FUNCTION_BLOCK RobotA26 EXTENDS KukaRobot
VAR_INPUT
	conveyorSafety : BOOL;
END_VAR
VAR_OUTPUT //from outputs array
	{warning disable C0195}
	taskID : TaskA26;
	param1 : INT; //position number (1..6)
	param2 : INT;
	
	strapSafetyOut : BOOL;
END_VAR
VAR_OUTPUT //from inputs array
	tool : SectionEnum := SectionEnum.SPACER_RECOLLECTOR;
	suspendedMaterial : STRING;
	
	completedTask : TaskA26;
	eoatDistance : INT;
	
	conveyorSafetyIn : BOOL;
END_VAR
VAR
	reservationEnum : SectionEnum;
	hmiTask : STRING;
	hmiTool : STRING;
END_VAR
(*
extends KukaRobot
	assigns descriptive labels to each IO group from the array
	additional section-specific methods to get/set IO groups
*)

(*
parameters - aliases to IO elements
command - full IO array
*)
{warning disable C0195}
SUPER^();

outputs[1] := taskID;
outputs[2] := param1;
outputs[3] := param2;

outputs[8].15 := conveyorSafety;

refreshParameters();

reservationEnum := reservation;
IF reservationEnum = SectionEnum.NULL_SECTION THEN
	hmiReservation := 'N/A';
ELSE
	hmiReservation := TO_STRING(reservationEnum);
END_IF

hmiTask := TO_STRING(taskID);
hmiTool := TO_STRING(tool);

{attribute 'monitoring' := 'call'}
PROPERTY Busy : BOOL
GET
VAR
	//emptyOutput : ARRAY[1..50] OF INT;
END_VAR
//Busy stays TRUE until outputs are cleared AND completed task has elapsed
//Ready is always inverse of Busy
refreshParameters();

Busy := taskID <> 0 OR completedTask <> 0;
END_GET
END_PROPERTY

METHOD clearCommand : BOOL
VAR_INPUT
END_VAR
SUPER^.clearCommand();

refreshParameters();
END_METHOD

{attribute 'monitoring' := 'call'}
PROPERTY Done : BOOL
GET
refreshParameters();

Done :=
	completedTask = taskID AND
	taskID <> 0 AND
	completedTask <> 0;
END_GET
END_PROPERTY

{attribute 'monitoring' := 'call'}
PROPERTY HoldMaterial : STRING
GET
HoldMaterial := suspendedMaterial;
END_GET
SET
suspendedMaterial := HoldMaterial;
END_SET
END_PROPERTY

{attribute 'monitoring' := 'call'}
PROPERTY Ready : BOOL
GET
refreshParameters();

Ready := taskID = 0 AND completedTask = 0 AND NOT error;
END_GET
END_PROPERTY

METHOD PRIVATE refreshParameters : BOOL
VAR_INPUT
END_VAR
{warning disable C0196}
taskID := outputs[1];
param1 := outputs[2];
param2 := outputs[3];

conveyorSafetyIn := inputs[4].15;
END_METHOD

METHOD setGroup : BOOL
VAR_INPUT
	group : INT;
	value : INT;
END_VAR
SUPER^.setGroup(group := group, value := value);

refreshParameters();
END_METHOD

METHOD setParameters : BOOL
VAR_INPUT
	newTaskID : INT;
	newParam1 : INT;
	newParam2 : INT;
	newXmm : INT;
	newYmm : INT;
	newZmm : INT;
	newAngle : INT;
	newStagingOccupancy : INT;
	newInsertionSuctionStatus : INT;
	newMagazineStatus : INT; //unused
	newInspectionValue : INT;
END_VAR
VAR_INPUT
	strapSafety : BOOL;
END_VAR
setGroup(group := 1, value := newTaskID);
setGroup(group := 2, value := newParam1);
setGroup(group := 3, value := newParam2);

refreshParameters();
END_METHOD

END_FUNCTION_BLOCK

(* stored: Version 1.1.0.1, ProductVersion 3.1.4024.11
   POU RobotA26: Id {33f267be-2dda-4e27-806e-968d4f9de821}, SpecialFunc None
   Folder Parameters: Id {23e176d2-b400-4b35-8de9-dcd6cb049883}
   Folder Properties: Id {bbdd7a8e-4dbc-4c64-8855-9dd2866686c7}
   Property Busy: Id {070ee2d5-320e-4280-bb50-110979219d3a}
   Get Get: Id {83b2a047-818c-40a4-95d3-5e235360971a}
   Method clearCommand: Id {091d3579-223c-434b-9fb6-186fe0d2bf80}
   Property Done: Id {916f564b-f94f-4aad-b35a-e00f859b03c2}
   Get Get: Id {b18c56f2-58a0-40c0-8d48-1befba46f464}
   Property HoldMaterial: Id {e46199aa-5e80-446c-8a9d-b18fe0d84c55}
   Get Get: Id {72d0c38c-5e67-447e-a759-65af0e5d6df4}
   Set Set: Id {29add2fc-91f4-4cb4-9802-2371b83f0154}
   Property Ready: Id {a7bc1c3c-de7a-4742-97b3-75cd5f5c7676}
   Get Get: Id {dc5879a6-f673-438e-868c-45288e7b4a3c}
   Method refreshParameters: Id {0b7f9e63-4312-456a-b2fa-3b911981f7a6}
   Method setGroup: Id {da0673d9-8bde-49d9-9378-89713e3e56b7}
   Method setParameters: Id {1ae0a962-c8e0-448b-bb16-693221bc5932} *)
